(* Schneider Machine Expert - Basic project Pockette, file version 1.2.0.0 *)

HARDWARE
  Cpu 0: TM221ME16T/G
  EthernetConfiguration: NetworkName=M221, IpAllocationMode=FixedAddress, IpAddress=0.0.0.0, SubnetMask=0.0.0.0
  SerialLineConfiguration: Baud=Baud19200, Parity=ParityEven, DataBits=DataBits8, StopBits=StopBits1, PhysicalMedium=PhysicalMediumRs485, TransmissionMode=TransmissionModeModbusRtu, SlaveId=1, Addressing=SlaveAddressing
  MastTask: UsePeriodScanMode=false, PeriodScan=100
  FastTask: Period=255
  CpuBehavior: StartingMode=StartInRun, AutoSaveRamOnEeprom=true, WatchdogPeriod=250

SYMBOLS  (address, symbol, comment, settings)

POU Nouveau POU
  (* SectionNumber=1, IsGrafcet=false *)

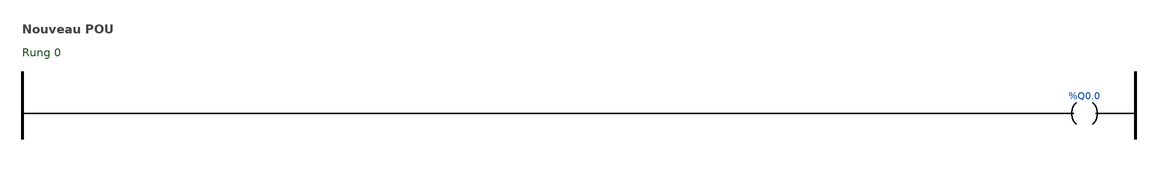

// Rung 0
  LD 1
  ST %Q0.0
  // as ST:
  //   %Q0.0 := TRUE;
